// TIA Portal V16 export
// export: Created 2026-06-19T08:38:32.7604192Z, ExportSetting WithDefaults, DisplayName Totally Integrated Automation Portal, DisplayVersion V16 Update 8, DisplayName TIA Portal Version Control Interface, DisplayVersion V16 Update 8, DisplayName TIA Portal Openness, DisplayVersion V16 Update 8, DisplayName SINAMICS Startdrive Advanced, DisplayVersion V16, DisplayName SINAMICS Startdrive G130, G150, S120, S150, SINAMICS MV, S210, DisplayVersion V16, DisplayName SINAMICS Startdrive G110M, G120, G120C, G120D, G120P, DisplayVersion V16, DisplayName STEP 7 Professional, DisplayVersion V16 Update 8, DisplayName STEP 7 Safety, DisplayVersion V16 Update 7, DisplayName WinCC Advanced, DisplayVersion V16 Update 8
Screen "画面_1"  800x480, Number=1
  ScreenLayer 
    Circle "圆_1" at 446,91 size 48x48
      RangeAppearanceAnimation "RangeAppearanceAnimation"
        tag Light
        0..0: back #dedbde, fore #181c31
        1..1: back #00ff00, fore #181c31
    Button "按钮_1" at 328,202 size 96x32  Mode=Text, TextOff="Text", TextOn="Text"
      on Press: SetBit(Tag := Button)
      on Release: ResetBit(Tag := Button)
    IOField "I/O 域_1" at 209,88 size 96x32  DataFormat=Decimal, FormatPattern=9999999, Mode=InOutput
    SymbolicIOField "符号 I/O 域_1" at 457,258 size 96x32  CountVisibleItems=3, Mode=InOutput, OnValue=1, TextOff="0", TextOn="1"
    TextField "文本域_1" at 516,73 size 41x20  Text="Text"
